TYPE ST_GovernorSerialAck :
STRUCT
	iPrefix			:	BYTE := 16#06;
	iStationNo		:	ARRAY [0..1] OF BYTE;
	iPCNo			:	ARRAY [0..1] OF BYTE;
END_STRUCT
END_TYPE

(* stored: Version 1.1.0.1, ProductVersion 3.1.4024.12
   DUT ST_GovernorSerialAck: Id {5382fc1f-8c5d-4fc9-8fdc-52e176374a95} *)
